// TIA Portal V20 export
DATA_BLOCK "EM_MotorData"   // DB188
// stored: MemoryReserve 100, Namespace Unit1
   VAR
      DR1_JROutPP_Left_X : LReal;
      DR2_JROutPP_Left_Z : LReal;
      DR3_JROutPP_Right_X : LReal;
      DR4_JROutPP_Right_Z : LReal;
      DR5_T_TapeAxis_X : LReal;
      DR6_T_TapeAxis_Y : LReal;
      DR7_S_TapeFixStage_X : LReal;
      DR8_S_TapeFixStage_C : LReal;
      DR9_S_Attachment_X : LReal;
      DR10_S_Attachment_Y : LReal;
      DR11_Thickness_Z : LReal;
      DR12_TrPP_Left_X : LReal;
      DR13_TrPP_Left_Y : LReal;
      DR14_TrPP_Left_Z : LReal;
      DR15_TrPP_Right_X : LReal;
      DR16_TrPP_Right_Y : LReal;
      DR17_TrPP_Right_Z : LReal;
      DR18_JRUloading_X : LReal;
      DR19_JRUloading_Z : LReal;
      DR20_JRUloading_C : LReal;
   END_VAR
BEGIN
END_DATA_BLOCK
